Staubli VAL3: DeleteAlarmFile.pgx

public program DeleteAlarmFile()
begin
  //删除报警文件
  if $fileExists("Usr://configs/sfty.dat")
    $delete("Usr://configs/sfty.dat")

  endIf


  if $fileExists("Usr://temp/pdrv.dat")

    $delete("Usr://temp/pdrv.dat")
  endIf












end
